% RSLogix 500 project ROTATION PROGRAM FOR PORTABLE BIN SCRUBBER_BAK000.RSS, saved by version 11.00.00.00 %
PROJECT "UNTITLED"    % processor: MicroLogix 1400 %

PROGRAM FILES
  LAD 2   20 rungs

DATA FILES
  O0 OUTPUT  6 elements
  I1 INPUT  8 elements
  S2 STATUS  66 elements
  B3 BINARY  1 elements
  T4 TIMER  1 elements
  C5 COUNTER  1 elements
  R6 CONTROL  1 elements
  N7 INTEGER  1 elements
  F8 FLOAT  1 elements

LADDER 2
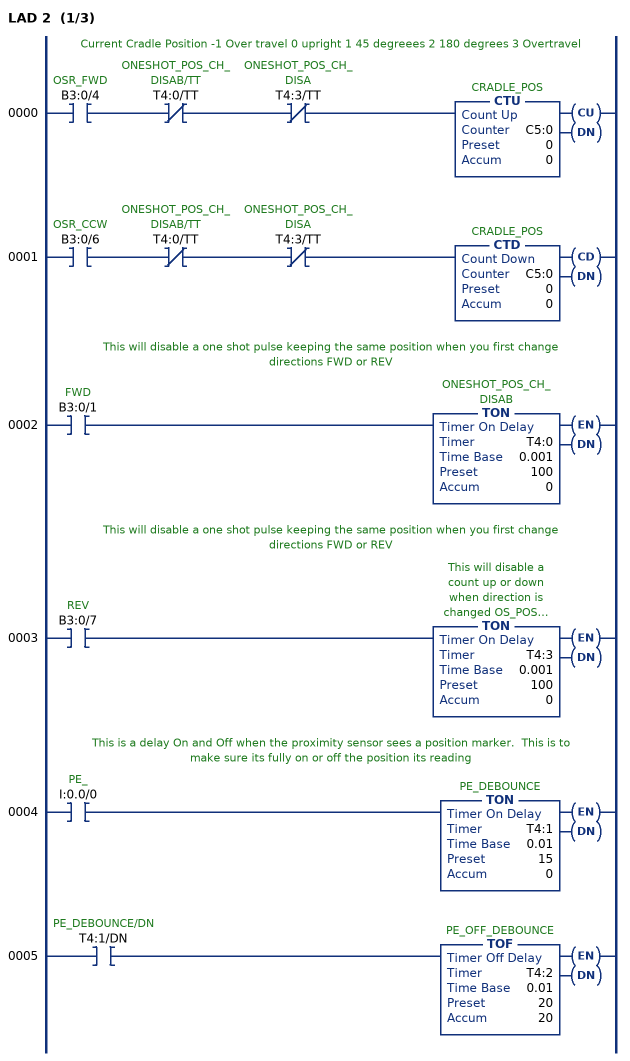
% Rung: 0 %  % edit flag set %
% Current Cradle Position -1 Over travel 0 upright 1 45 degreees 2 180 degrees 3 Overtravel %
SOR XIC B3:0/4 XIO T4:0/TT XIO T4:3/TT CTU C5:0 0 0 EOR
%   B3:0/4  OSR_FWD %
%   T4:0  ONESHOT_POS_CH_DISAB %
%   T4:3/TT  ONESHOT_POS_CH_DISA %
%   C5:0  CRADLE_POS %
% Rung: 1 %  % edit flag set %
SOR XIC B3:0/6 XIO T4:0/TT XIO T4:3/TT CTD C5:0 0 0 EOR
%   B3:0/6  OSR_CCW %
%   T4:0  ONESHOT_POS_CH_DISAB %
%   T4:3/TT  ONESHOT_POS_CH_DISA %
%   C5:0  CRADLE_POS %
% Rung: 2 %  % edit flag set %
% This will disable a one shot pulse keeping the same position when you first change directions FWD or REV %
SOR XIC B3:0/1 TON T4:0 0.001 100 0 EOR
%   B3:0/1  FWD %
%   T4:0  ONESHOT_POS_CH_DISAB %
% Rung: 3 %  % edit flag set %
% This will disable a one shot pulse keeping the same position when you first change directions FWD or REV %
SOR XIC B3:0/7 TON T4:3 0.001 100 0 EOR
%   B3:0/7  REV %
%   T4:3  OS_POS_CHANGE_DISABL  "This will disable a count up or down when direction is changed" %
% Rung: 4 %  % edit flag set %
% This is a delay On and Off when the proximity sensor sees a position marker.  This is to make sure its fully on or off the position its reading %
SOR XIC I:0.0/0 TON T4:1 0.01 15 0 EOR
%   I:0.0/0  PE_ %
%   T4:1  PE_DEBOUNCE %
% Rung: 5 %  % edit flag set %
SOR XIC T4:1/DN TOF T4:2 0.01 20 20 EOR
%   T4:1  PE_DEBOUNCE %
%   T4:2  PE_OFF_DEBOUNCE %

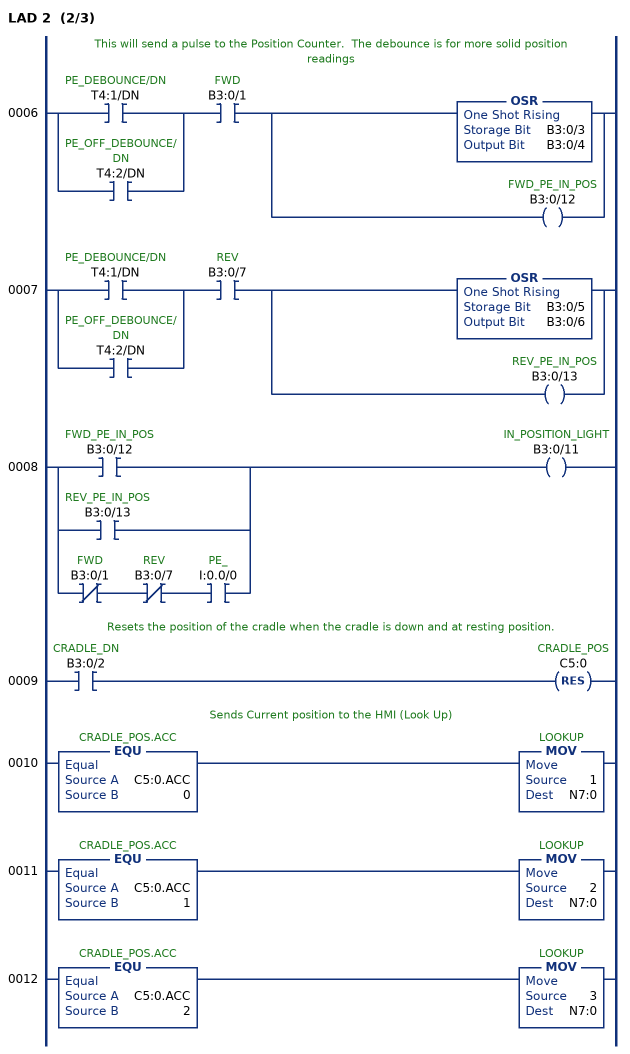
% Rung: 6 %  % edit flag set %
% This will send a pulse to the Position Counter.  The debounce is for more solid position readings %
SOR BST XIC T4:1/DN NXB XIC T4:2/DN BND XIC B3:0/1 BST OSR B3:0/3 B3:0/4 NXB OTE B3:0/12 BND EOR
%   T4:1  PE_DEBOUNCE %
%   T4:2  PE_OFF_DEBOUNCE %
%   B3:0/1  FWD %
%   B3:0/4  OSR_FWD %
%   B3:0/12  FWD_PE_IN_POS %
% Rung: 7 %  % edit flag set %
SOR BST XIC T4:1/DN NXB XIC T4:2/DN BND XIC B3:0/7 BST OSR B3:0/5 B3:0/6 NXB OTE B3:0/13 BND EOR
%   T4:1  PE_DEBOUNCE %
%   T4:2  PE_OFF_DEBOUNCE %
%   B3:0/7  REV %
%   B3:0/6  OSR_CCW %
%   B3:0/13  REV_PE_IN_POS %
% Rung: 8 %  % edit flag set %
SOR BST XIC B3:0/12 NXB BST XIC B3:0/13 NXB XIO B3:0/1 XIO B3:0/7 XIC I:0.0/0 BND BND OTE B3:0/11 EOR
%   B3:0/12  FWD_PE_IN_POS %
%   B3:0/13  REV_PE_IN_POS %
%   B3:0/1  FWD %
%   B3:0/7  REV %
%   I:0.0/0  PE_ %
%   B3:0/11  IN_POSITION_LIGHT %
% Rung: 9 %  % edit flag set %
% Resets the position of the cradle when the cradle is down and at resting position. %
SOR XIC B3:0/2 RES C5:0 EOR
%   B3:0/2  CRADLE_DN %
%   C5:0  CRADLE_POS %
% Rung: 10 %  % edit flag set %
% Sends Current position to the HMI (Look Up) %
SOR EQU C5:0.ACC 0 MOV 1 N7:0 EOR
%   C5:0  CRADLE_POS %
%   N7:0  LOOKUP %
% Rung: 11 %  % edit flag set %
SOR EQU C5:0.ACC 1 MOV 2 N7:0 EOR
%   C5:0  CRADLE_POS %
%   N7:0  LOOKUP %
% Rung: 12 %  % edit flag set %
SOR EQU C5:0.ACC 2 MOV 3 N7:0 EOR
%   C5:0  CRADLE_POS %
%   N7:0  LOOKUP %

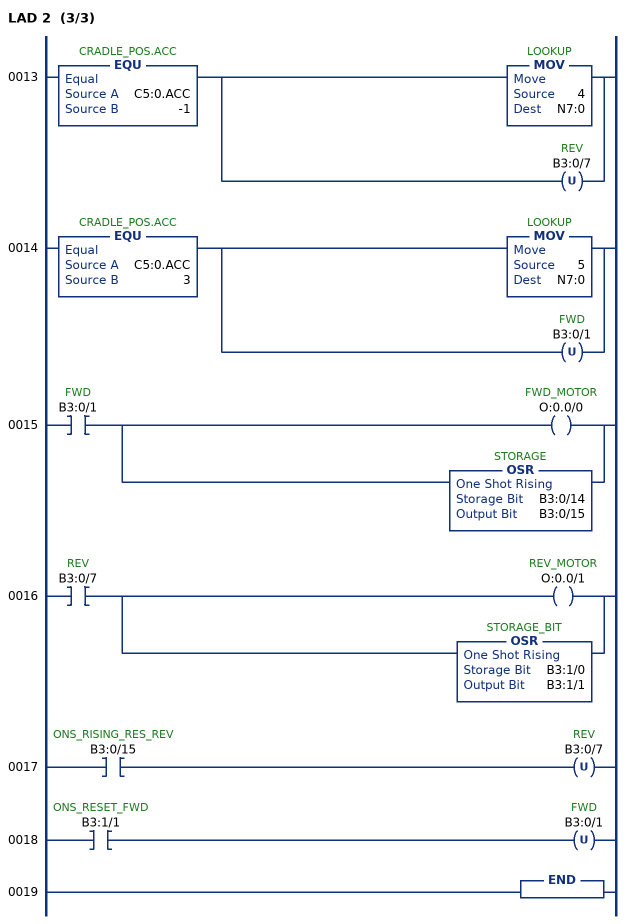
% Rung: 13 %  % edit flag set %
SOR EQU C5:0.ACC -1 BST MOV 4 N7:0 NXB OTU B3:0/7 BND EOR
%   C5:0  CRADLE_POS %
%   N7:0  LOOKUP %
%   B3:0/7  REV %
% Rung: 14 %  % edit flag set %
SOR EQU C5:0.ACC 3 BST MOV 5 N7:0 NXB OTU B3:0/1 BND EOR
%   C5:0  CRADLE_POS %
%   N7:0  LOOKUP %
%   B3:0/1  FWD %
% Rung: 15 %  % edit flag set %
SOR XIC B3:0/1 BST OTE O:0.0/0 NXB OSR B3:0/14 B3:0/15 BND EOR
%   B3:0/1  FWD %
%   O:0.0/0  FWD_MOTOR %
%   B3:0/14  STORAGE %
%   B3:0/15  ONS_RISING_RES_REV %
% Rung: 16 %  % edit flag set %
SOR XIC B3:0/7 BST OTE O:0.0/1 NXB OSR B3:1/0 B3:1/1 BND EOR
%   B3:0/7  REV %
%   O:0.0/1  REV_MOTOR %
%   B3:1/0  STORAGE_BIT %
%   B3:1/1  ONS_RESET_FWD %
% Rung: 17 %  % edit flag set %
SOR XIC B3:0/15 OTU B3:0/7 EOR
%   B3:0/15  ONS_RISING_RES_REV %
%   B3:0/7  REV %
% Rung: 18 %  % edit flag set %
SOR XIC B3:1/1 OTU B3:0/1 EOR
%   B3:1/1  ONS_RESET_FWD %
%   B3:0/1  FWD %
% Rung: 19 %
SOR END EOR
